(* IEC 61131-3 sources: weg-scada/M241_Bridge, 5 files *)

(* ---- POU_Diagnostics.st ---- *)
(*
  POU_Diagnostics - OPCIONAL

  Este programa es OPCIONAL. El M241 funciona como bridge transparente
  sin necesidad de programacion. Solo agregar este POU si se quiere
  monitorear el estado de comunicacion desde el PLC.

  Importar en Machine Expert: Project > Import > PLCOpen XML
  Asignar a MAST task si se usa.
*)

PROGRAM POU_Diagnostics
VAR
    (* Timers para detectar perdida de comunicacion *)
    tSSW1_Watchdog : TON;
    tSSW2_Watchdog : TON;

    (* Valores anteriores para detectar cambios *)
    wSSW1_PrevStatus : WORD := 16#FFFF;
    wSSW2_PrevStatus : WORD := 16#FFFF;

    (* Comunicacion OK flags *)
    bSSW1_Alive : BOOL;
    bSSW2_Alive : BOOL;

    (* Contadores de error *)
    udiSSW1_Errors : UDINT;
    udiSSW2_Errors : UDINT;

    (* LED output para diagnostico - usar salida digital del M241 *)
    bLED_AllOK     AT %QX0.0 : BOOL;  (* Q0 = Todos los esclavos OK *)
    bLED_SSW1_Fail AT %QX0.1 : BOOL;  (* Q1 = SSW1 sin comunicacion *)
    bLED_SSW2_Fail AT %QX0.2 : BOOL;  (* Q2 = SSW2 sin comunicacion *)
END_VAR

(* Detectar si SSW900 #1 esta respondiendo *)
(* Si el status word cambia, el esclavo esta vivo *)
IF GVL_SSW900.SSW1_StatusWord <> wSSW1_PrevStatus THEN
    wSSW1_PrevStatus := GVL_SSW900.SSW1_StatusWord;
    bSSW1_Alive := TRUE;
    tSSW1_Watchdog(IN := FALSE);  (* Reset timer *)
END_IF

tSSW1_Watchdog(IN := TRUE, PT := T#10S);
IF tSSW1_Watchdog.Q THEN
    bSSW1_Alive := FALSE;
    udiSSW1_Errors := udiSSW1_Errors + 1;
    tSSW1_Watchdog(IN := FALSE);
END_IF

(* Detectar si SSW900 #2 esta respondiendo *)
IF GVL_SSW900.SSW2_StatusWord <> wSSW2_PrevStatus THEN
    wSSW2_PrevStatus := GVL_SSW900.SSW2_StatusWord;
    bSSW2_Alive := TRUE;
    tSSW2_Watchdog(IN := FALSE);
END_IF

tSSW2_Watchdog(IN := TRUE, PT := T#10S);
IF tSSW2_Watchdog.Q THEN
    bSSW2_Alive := FALSE;
    udiSSW2_Errors := udiSSW2_Errors + 1;
    tSSW2_Watchdog(IN := FALSE);
END_IF

(* Actualizar variables globales *)
GVL_SSW900.SSW1_CommOK := bSSW1_Alive;
GVL_SSW900.SSW2_CommOK := bSSW2_Alive;
GVL_SSW900.SSW1_CommErrors := udiSSW1_Errors;
GVL_SSW900.SSW2_CommErrors := udiSSW2_Errors;

(* LEDs de diagnostico *)
bLED_AllOK := bSSW1_Alive AND bSSW2_Alive;
bLED_SSW1_Fail := NOT bSSW1_Alive;
bLED_SSW2_Fail := NOT bSSW2_Alive;

(* ---- WEG_Banner_Trending.st ---- *)
// ============================================================================
// WEG ALARM BANNER + TRENDING SUPPORT
// Single scrolling banner showing active faults from all 8 devices
// Trending buffer for WebVisu Trend element
// ============================================================================

// ============================================================================
// GVL: GVL_Banner (add to existing GVL_HMI or create separate)
// ============================================================================

{attribute 'qualified_only'}
VAR_GLOBAL

    // ---- Alarm Banner ----
    sBannerText         : STRING(255);      // Current text displayed in banner
    sBannerFull         : STRING(255);      // Full concatenated alarm string
    bBannerBlink        : BOOL;             // Blink flag for banner background
    iBannerColor        : INT;              // 0=No alarms(green), 1=Warning(yellow), 2=Fault(red)
    bHasFaults          : BOOL;             // At least one fault active

    // ---- Trending Data (WebVisu Trend uses these directly) ----
    // CFW900 Currents
    rTrend_CFW1_Current : REAL;
    rTrend_CFW2_Current : REAL;
    rTrend_CFW3_Current : REAL;
    rTrend_CFW4_Current : REAL;

    // CFW900 Frequencies
    rTrend_CFW1_Freq    : REAL;
    rTrend_CFW2_Freq    : REAL;
    rTrend_CFW3_Freq    : REAL;
    rTrend_CFW4_Freq    : REAL;

    // SSW900 Currents
    rTrend_SSW1_Current : REAL;
    rTrend_SSW2_Current : REAL;
    rTrend_SSW3_Current : REAL;
    rTrend_SSW4_Current : REAL;

END_VAR

// ============================================================================
// PROGRAM: PRG_AlarmBanner
// Builds a single scrolling text with all active faults
// Task: MAST
// ============================================================================

PROGRAM PRG_AlarmBanner
VAR
    i               : INT;
    sTemp           : STRING(255);
    iFaultCount     : INT;

    // Scroll control
    iScrollPos      : INT := 0;
    iScrollLen      : INT;
    tScrollTimer    : TON;
    tBlinkTimer     : TON;
    bBlinkState     : BOOL;

    // Rotation: cycle through faults one at a time
    iDisplayIndex   : INT := 0;         // Which fault to show (0..iFaultCount-1)
    tRotateTimer    : TON;
    aFaultMessages  : ARRAY[0..7] OF STRING(80);
    iFaultTotal     : INT;
END_VAR

// =========================================
// STEP 1: Collect all active faults
// =========================================
iFaultTotal := 0;

// Check CFW900 devices
FOR i := 1 TO 4 DO
    IF GVL_WEG.stCFW900[i].bFault THEN
        aFaultMessages[iFaultTotal] := CONCAT(
            CONCAT('CFW900#', INT_TO_STRING(i)),
            CONCAT(': ', FC_CFW900_FaultText(GVL_WEG.stCFW900[i].wFaultCode))
        );
        iFaultTotal := iFaultTotal + 1;

    ELSIF NOT GVL_WEG.stCFW900[i].bOnline AND GVL_WEG.stCFW900[i].uiCommErrCount > 5 THEN
        aFaultMessages[iFaultTotal] := CONCAT('CFW900#', CONCAT(INT_TO_STRING(i), ': COMM LOST'));
        iFaultTotal := iFaultTotal + 1;
    END_IF;
END_FOR;

// Check SSW900 devices
FOR i := 1 TO 4 DO
    IF GVL_WEG.stSSW900[i].bFault THEN
        aFaultMessages[iFaultTotal] := CONCAT(
            CONCAT('SSW900#', INT_TO_STRING(i)),
            CONCAT(': ', FC_SSW900_FaultText(GVL_WEG.stSSW900[i].wFaultCode))
        );
        iFaultTotal := iFaultTotal + 1;

    ELSIF NOT GVL_WEG.stSSW900[i].bOnline AND GVL_WEG.stSSW900[i].uiCommErrCount > 5 THEN
        aFaultMessages[iFaultTotal] := CONCAT('SSW900#', CONCAT(INT_TO_STRING(i), ': COMM LOST'));
        iFaultTotal := iFaultTotal + 1;
    END_IF;
END_FOR;

// =========================================
// STEP 2: Update banner state
// =========================================
GVL_Banner.bHasFaults := (iFaultTotal > 0);

IF iFaultTotal = 0 THEN
    // No faults - show OK message
    GVL_Banner.sBannerText := 'SYSTEM OK - All drives operating normally';
    GVL_Banner.iBannerColor := 0;       // Green
    GVL_Banner.bBannerBlink := FALSE;
    iDisplayIndex := 0;

ELSIF iFaultTotal = 1 THEN
    // Single fault - show it fixed (no rotation needed)
    GVL_Banner.sBannerText := CONCAT('!! ', CONCAT(aFaultMessages[0], ' !!'));
    GVL_Banner.iBannerColor := 2;       // Red
    GVL_Banner.bBannerBlink := TRUE;

ELSE
    // Multiple faults - rotate display every 3 seconds
    tRotateTimer(IN := TRUE, PT := T#3S);
    IF tRotateTimer.Q THEN
        tRotateTimer(IN := FALSE);
        iDisplayIndex := iDisplayIndex + 1;
        IF iDisplayIndex >= iFaultTotal THEN
            iDisplayIndex := 0;
        END_IF;
    END_IF;

    // Build display: "!! [2/3] CFW900#1: F002 Overcurrent !!"
    GVL_Banner.sBannerText := CONCAT(
        CONCAT('!! [', CONCAT(INT_TO_STRING(iDisplayIndex + 1), CONCAT('/', INT_TO_STRING(iFaultTotal)))),
        CONCAT('] ', CONCAT(aFaultMessages[iDisplayIndex], ' !!'))
    );
    GVL_Banner.iBannerColor := 2;       // Red
    GVL_Banner.bBannerBlink := TRUE;

END_IF;

// =========================================
// STEP 3: Blink control (500ms toggle)
// =========================================
tBlinkTimer(IN := NOT tBlinkTimer.Q, PT := T#500MS);
IF tBlinkTimer.Q THEN
    bBlinkState := NOT bBlinkState;
END_IF;

IF GVL_Banner.bBannerBlink THEN
    GVL_Banner.bBannerBlink := bBlinkState;    // Toggle for HMI animation
END_IF;

// ============================================================================
// PROGRAM: PRG_Trending
// Copies monitoring data to trending variables
// Task: MAST
// ============================================================================

PROGRAM PRG_Trending
VAR
END_VAR

// CFW900 Currents
GVL_Banner.rTrend_CFW1_Current := GVL_WEG.stCFW900[1].rOutputCurrent;
GVL_Banner.rTrend_CFW2_Current := GVL_WEG.stCFW900[2].rOutputCurrent;
GVL_Banner.rTrend_CFW3_Current := GVL_WEG.stCFW900[3].rOutputCurrent;
GVL_Banner.rTrend_CFW4_Current := GVL_WEG.stCFW900[4].rOutputCurrent;

// CFW900 Frequencies
GVL_Banner.rTrend_CFW1_Freq := GVL_WEG.stCFW900[1].rOutputFreq;
GVL_Banner.rTrend_CFW2_Freq := GVL_WEG.stCFW900[2].rOutputFreq;
GVL_Banner.rTrend_CFW3_Freq := GVL_WEG.stCFW900[3].rOutputFreq;
GVL_Banner.rTrend_CFW4_Freq := GVL_WEG.stCFW900[4].rOutputFreq;

// SSW900 Currents
GVL_Banner.rTrend_SSW1_Current := GVL_WEG.stSSW900[1].rMotorCurrent;
GVL_Banner.rTrend_SSW2_Current := GVL_WEG.stSSW900[2].rMotorCurrent;
GVL_Banner.rTrend_SSW3_Current := GVL_WEG.stSSW900[3].rMotorCurrent;
GVL_Banner.rTrend_SSW4_Current := GVL_WEG.stSSW900[4].rMotorCurrent;

(* ---- WEG_DataLog_Voltage.st ---- *)
// ============================================================================
// WEG DATA LOGGING (SD Card) + VOLTAGE EMPHASIS
// Exports CSV to M241 SD card + enhanced voltage monitoring
// Libraries required: FileIO, SysFile, SysTimeRtc, CAA File
// ============================================================================

// ============================================================================
// GVL: GVL_DataLog
// ============================================================================

{attribute 'qualified_only'}
VAR_GLOBAL

    // ---- Data Logging Control ----
    bLogEnabled         : BOOL := TRUE;     // Enable/disable logging from HMI
    bLogActive          : BOOL;             // Logging is running
    bLogError           : BOOL;             // File error occurred
    sLogStatus          : STRING(60);       // Status message for HMI
    iLogInterval        : INT := 5;         // Log interval in seconds (adjustable from HMI)
    ulRecordCount       : UDINT;            // Total records written

    // ---- File Management ----
    bNewFileDaily       : BOOL := TRUE;     // Create new file each day
    sCurrentFileName    : STRING(80);       // Current log file name
    bSDCardPresent      : BOOL;             // SD card detected
    ulFileSizeKB        : UDINT;            // Current file size

    // ---- Manual Export Trigger ----
    bExportSnapshot     : BOOL;             // Trigger single snapshot from HMI
    bExportDone         : BOOL;             // Snapshot saved confirmation

    // ---- Voltage Monitoring (Enhanced) ----
    // CFW900 Voltages
    stCFW_Voltage       : ARRAY[1..4] OF ST_VoltageMonitor;

    // SSW900 Voltages
    stSSW_Voltage       : ARRAY[1..4] OF ST_VoltageMonitor;

    // Voltage Alarms
    bVoltageAlarmActive : BOOL;             // Any voltage alarm
    iVoltageAlarmCount  : INT;

    // Voltage Thresholds (adjustable from HMI)
    rCFW_DCBus_High     : REAL := 750.0;    // DC Bus overvoltage threshold (V)
    rCFW_DCBus_Low      : REAL := 350.0;    // DC Bus undervoltage threshold (V)
    rSSW_Motor_High     : REAL := 480.0;    // Motor overvoltage threshold (V)
    rSSW_Motor_Low      : REAL := 400.0;    // Motor undervoltage threshold (V)
    rSSW_Imbalance_Max  : REAL := 5.0;      // Max voltage imbalance (%) between SSW units

    // Trending Voltage
    rTrend_CFW1_DCVoltage : REAL;
    rTrend_CFW2_DCVoltage : REAL;
    rTrend_CFW3_DCVoltage : REAL;
    rTrend_CFW4_DCVoltage : REAL;
    rTrend_SSW1_Voltage   : REAL;
    rTrend_SSW2_Voltage   : REAL;
    rTrend_SSW3_Voltage   : REAL;
    rTrend_SSW4_Voltage   : REAL;

END_VAR

// ============================================================================
// DUT: ST_VoltageMonitor
// ============================================================================

TYPE ST_VoltageMonitor :
STRUCT
    rVoltageNow     : REAL;         // Current voltage reading
    rVoltageMin     : REAL;         // Minimum since reset
    rVoltageMax     : REAL;         // Maximum since reset
    rVoltageAvg     : REAL;         // Running average

    // Alarms
    bOvervoltage    : BOOL;         // Above high threshold
    bUndervoltage   : BOOL;         // Below low threshold
    bAlarm          : BOOL;         // Any voltage alarm

    // Stats
    rDeviation      : REAL;         // Deviation from average (%)
    ulSampleCount   : UDINT;        // Samples for average calc
    rAccumulator    : LREAL;        // Sum for average (internal)
END_STRUCT
END_TYPE

// ============================================================================
// PROGRAM: PRG_VoltageMonitor
// Enhanced voltage tracking with min/max/avg and alarms
// Task: MAST
// ============================================================================

PROGRAM PRG_VoltageMonitor
VAR
    i               : INT;
    rAvgSSW         : REAL;         // Average voltage across all SSW units
    iOnlineSSW      : INT;
    bFirstScan      : BOOL := TRUE;
END_VAR

// =========================================
// Initialize min/max on first scan
// =========================================
IF bFirstScan THEN
    FOR i := 1 TO 4 DO
        GVL_DataLog.stCFW_Voltage[i].rVoltageMin := 9999.0;
        GVL_DataLog.stCFW_Voltage[i].rVoltageMax := 0.0;
        GVL_DataLog.stSSW_Voltage[i].rVoltageMin := 9999.0;
        GVL_DataLog.stSSW_Voltage[i].rVoltageMax := 0.0;
    END_FOR;
    bFirstScan := FALSE;
END_IF;

// =========================================
// CFW900: DC Bus Voltage monitoring
// =========================================
GVL_DataLog.iVoltageAlarmCount := 0;

FOR i := 1 TO 4 DO
    IF GVL_WEG.stCFW900[i].bOnline THEN

        GVL_DataLog.stCFW_Voltage[i].rVoltageNow := GVL_WEG.stCFW900[i].rDCBusVoltage;

        // Min / Max
        IF GVL_DataLog.stCFW_Voltage[i].rVoltageNow < GVL_DataLog.stCFW_Voltage[i].rVoltageMin THEN
            GVL_DataLog.stCFW_Voltage[i].rVoltageMin := GVL_DataLog.stCFW_Voltage[i].rVoltageNow;
        END_IF;
        IF GVL_DataLog.stCFW_Voltage[i].rVoltageNow > GVL_DataLog.stCFW_Voltage[i].rVoltageMax THEN
            GVL_DataLog.stCFW_Voltage[i].rVoltageMax := GVL_DataLog.stCFW_Voltage[i].rVoltageNow;
        END_IF;

        // Running average
        GVL_DataLog.stCFW_Voltage[i].ulSampleCount := GVL_DataLog.stCFW_Voltage[i].ulSampleCount + 1;
        GVL_DataLog.stCFW_Voltage[i].rAccumulator := GVL_DataLog.stCFW_Voltage[i].rAccumulator +
            REAL_TO_LREAL(GVL_DataLog.stCFW_Voltage[i].rVoltageNow);

        IF GVL_DataLog.stCFW_Voltage[i].ulSampleCount > 0 THEN
            GVL_DataLog.stCFW_Voltage[i].rVoltageAvg := LREAL_TO_REAL(
                GVL_DataLog.stCFW_Voltage[i].rAccumulator /
                UDINT_TO_LREAL(GVL_DataLog.stCFW_Voltage[i].ulSampleCount)
            );
        END_IF;

        // Overvoltage / Undervoltage alarms
        GVL_DataLog.stCFW_Voltage[i].bOvervoltage :=
            GVL_DataLog.stCFW_Voltage[i].rVoltageNow > GVL_DataLog.rCFW_DCBus_High;
        GVL_DataLog.stCFW_Voltage[i].bUndervoltage :=
            GVL_DataLog.stCFW_Voltage[i].rVoltageNow < GVL_DataLog.rCFW_DCBus_Low;
        GVL_DataLog.stCFW_Voltage[i].bAlarm :=
            GVL_DataLog.stCFW_Voltage[i].bOvervoltage OR GVL_DataLog.stCFW_Voltage[i].bUndervoltage;

        IF GVL_DataLog.stCFW_Voltage[i].bAlarm THEN
            GVL_DataLog.iVoltageAlarmCount := GVL_DataLog.iVoltageAlarmCount + 1;
        END_IF;

    END_IF;
END_FOR;

// =========================================
// SSW900: Motor Voltage monitoring
// =========================================
rAvgSSW := 0.0;
iOnlineSSW := 0;

FOR i := 1 TO 4 DO
    IF GVL_WEG.stSSW900[i].bOnline THEN

        GVL_DataLog.stSSW_Voltage[i].rVoltageNow := GVL_WEG.stSSW900[i].rMotorVoltage;

        // Min / Max
        IF GVL_DataLog.stSSW_Voltage[i].rVoltageNow < GVL_DataLog.stSSW_Voltage[i].rVoltageMin THEN
            GVL_DataLog.stSSW_Voltage[i].rVoltageMin := GVL_DataLog.stSSW_Voltage[i].rVoltageNow;
        END_IF;
        IF GVL_DataLog.stSSW_Voltage[i].rVoltageNow > GVL_DataLog.stSSW_Voltage[i].rVoltageMax THEN
            GVL_DataLog.stSSW_Voltage[i].rVoltageMax := GVL_DataLog.stSSW_Voltage[i].rVoltageNow;
        END_IF;

        // Running average
        GVL_DataLog.stSSW_Voltage[i].ulSampleCount := GVL_DataLog.stSSW_Voltage[i].ulSampleCount + 1;
        GVL_DataLog.stSSW_Voltage[i].rAccumulator := GVL_DataLog.stSSW_Voltage[i].rAccumulator +
            REAL_TO_LREAL(GVL_DataLog.stSSW_Voltage[i].rVoltageNow);

        IF GVL_DataLog.stSSW_Voltage[i].ulSampleCount > 0 THEN
            GVL_DataLog.stSSW_Voltage[i].rVoltageAvg := LREAL_TO_REAL(
                GVL_DataLog.stSSW_Voltage[i].rAccumulator /
                UDINT_TO_LREAL(GVL_DataLog.stSSW_Voltage[i].ulSampleCount)
            );
        END_IF;

        // Overvoltage / Undervoltage alarms
        GVL_DataLog.stSSW_Voltage[i].bOvervoltage :=
            GVL_DataLog.stSSW_Voltage[i].rVoltageNow > GVL_DataLog.rSSW_Motor_High;
        GVL_DataLog.stSSW_Voltage[i].bUndervoltage :=
            GVL_DataLog.stSSW_Voltage[i].rVoltageNow < GVL_DataLog.rSSW_Motor_Low;
        GVL_DataLog.stSSW_Voltage[i].bAlarm :=
            GVL_DataLog.stSSW_Voltage[i].bOvervoltage OR GVL_DataLog.stSSW_Voltage[i].bUndervoltage;

        IF GVL_DataLog.stSSW_Voltage[i].bAlarm THEN
            GVL_DataLog.iVoltageAlarmCount := GVL_DataLog.iVoltageAlarmCount + 1;
        END_IF;

        // Accumulate for imbalance calculation
        rAvgSSW := rAvgSSW + GVL_DataLog.stSSW_Voltage[i].rVoltageNow;
        iOnlineSSW := iOnlineSSW + 1;

    END_IF;
END_FOR;

// =========================================
// SSW900: Voltage imbalance detection
// =========================================
IF iOnlineSSW >= 2 THEN
    rAvgSSW := rAvgSSW / INT_TO_REAL(iOnlineSSW);

    FOR i := 1 TO 4 DO
        IF GVL_WEG.stSSW900[i].bOnline AND rAvgSSW > 0.0 THEN
            GVL_DataLog.stSSW_Voltage[i].rDeviation :=
                ABS(GVL_DataLog.stSSW_Voltage[i].rVoltageNow - rAvgSSW) / rAvgSSW * 100.0;

            // Flag if deviation exceeds threshold
            IF GVL_DataLog.stSSW_Voltage[i].rDeviation > GVL_DataLog.rSSW_Imbalance_Max THEN
                GVL_DataLog.stSSW_Voltage[i].bAlarm := TRUE;
                GVL_DataLog.iVoltageAlarmCount := GVL_DataLog.iVoltageAlarmCount + 1;
            END_IF;
        END_IF;
    END_FOR;
END_IF;

GVL_DataLog.bVoltageAlarmActive := (GVL_DataLog.iVoltageAlarmCount > 0);

// =========================================
// Update trending voltage variables
// =========================================
GVL_DataLog.rTrend_CFW1_DCVoltage := GVL_DataLog.stCFW_Voltage[1].rVoltageNow;
GVL_DataLog.rTrend_CFW2_DCVoltage := GVL_DataLog.stCFW_Voltage[2].rVoltageNow;
GVL_DataLog.rTrend_CFW3_DCVoltage := GVL_DataLog.stCFW_Voltage[3].rVoltageNow;
GVL_DataLog.rTrend_CFW4_DCVoltage := GVL_DataLog.stCFW_Voltage[4].rVoltageNow;
GVL_DataLog.rTrend_SSW1_Voltage   := GVL_DataLog.stSSW_Voltage[1].rVoltageNow;
GVL_DataLog.rTrend_SSW2_Voltage   := GVL_DataLog.stSSW_Voltage[2].rVoltageNow;
GVL_DataLog.rTrend_SSW3_Voltage   := GVL_DataLog.stSSW_Voltage[3].rVoltageNow;
GVL_DataLog.rTrend_SSW4_Voltage   := GVL_DataLog.stSSW_Voltage[4].rVoltageNow;

// ============================================================================
// PROGRAM: PRG_DataLogger
// Writes CSV records to M241 SD card
// Task: MAST
// Libraries: CAA File (SysFile), SysTimeRtc
// ============================================================================

PROGRAM PRG_DataLogger
VAR
    // State machine
    iStep           : INT := 0;

    // Timer for log interval
    tLogInterval    : TON;
    tLogPT          : TIME;

    // File handling
    hFile           : CAA.FILE.FILE_HANDLE := CAA.FILE.INVALID_HANDLE;
    fbFileOpen      : CAA.FILE.Open;
    fbFileWrite     : CAA.FILE.Write;
    fbFileClose     : CAA.FILE.Close;

    // Date/Time
    dtCurrent       : DT;
    stTime          : TIMESTRUCT;
    sDate           : STRING(12);
    sTime           : STRING(10);
    sFileName       : STRING(80);

    // CSV building
    sCSVHeader      : STRING(255);
    sCSVLine        : STRING(255);
    sCSVLine2       : STRING(255);      // Continuation (long line)
    sTemp           : STRING(20);

    // State tracking
    iLastDay        : INT := -1;
    bHeaderWritten  : BOOL;
    bWriteError     : BOOL;
    i               : INT;
END_VAR

// =========================================
// Build log interval from HMI setting
// =========================================
tLogPT := INT_TO_TIME(GVL_DataLog.iLogInterval * 1000);

CASE iStep OF

    0: // ---- CHECK IF LOGGING ENABLED ----
        IF NOT GVL_DataLog.bLogEnabled THEN
            GVL_DataLog.bLogActive := FALSE;
            GVL_DataLog.sLogStatus := 'Logging disabled';
            RETURN;
        END_IF;

        GVL_DataLog.bLogActive := TRUE;
        iStep := 5;

    5: // ---- GET CURRENT DATE/TIME ----
        dtCurrent := GET_DATETIME();
        stTime := DT_TO_TIMESTRUCT(dtCurrent);

        // Build date string YYYY-MM-DD
        sDate := CONCAT(
            CONCAT(INT_TO_STRING(stTime.wYear), '-'),
            CONCAT(FC_PadZero(stTime.wMonth), CONCAT('-', FC_PadZero(stTime.wDay)))
        );

        // Build time string HH:MM:SS
        sTime := CONCAT(
            CONCAT(FC_PadZero(stTime.wHour), ':'),
            CONCAT(FC_PadZero(stTime.wMinute), CONCAT(':', FC_PadZero(stTime.wSecond)))
        );

        // Build filename: /sd0/WEG_LOG_2026-03-30.csv
        sFileName := CONCAT('/sd0/WEG_LOG_', CONCAT(sDate, '.csv'));
        GVL_DataLog.sCurrentFileName := sFileName;

        // Check if new day = new file
        IF INT_TO_INT(stTime.wDay) <> iLastDay THEN
            iLastDay := INT_TO_INT(stTime.wDay);
            bHeaderWritten := FALSE;
        END_IF;

        iStep := 10;

    10: // ---- WAIT FOR LOG INTERVAL ----
        tLogInterval(IN := TRUE, PT := tLogPT);

        // Also check for manual snapshot trigger
        IF tLogInterval.Q OR GVL_DataLog.bExportSnapshot THEN
            tLogInterval(IN := FALSE);
            GVL_DataLog.bExportSnapshot := FALSE;
            iStep := 20;
        END_IF;

    20: // ---- OPEN FILE (APPEND MODE) ----
        fbFileOpen(
            sFileName   := sFileName,
            eFileMode   := CAA.FILE.MODE.MRDWR,    // Read/Write (append)
            xExclusive  := FALSE
        );

        IF fbFileOpen.xDone THEN
            hFile := fbFileOpen.hFile;
            GVL_DataLog.bLogError := FALSE;

            IF NOT bHeaderWritten THEN
                iStep := 25;    // Write header first
            ELSE
                iStep := 30;    // Skip to data
            END_IF;

        ELSIF fbFileOpen.xError THEN
            // File might not exist, try create
            GVL_DataLog.bLogError := TRUE;
            GVL_DataLog.sLogStatus := 'SD Card error - check card';
            iStep := 10;
        END_IF;

    25: // ---- WRITE CSV HEADER ----
        sCSVHeader := 'DateTime,';
        sCSVHeader := CONCAT(sCSVHeader, 'CFW1_A,CFW1_Hz,CFW1_VDC,CFW1_Torq,CFW1_RPM,CFW1_Sts,');
        sCSVHeader := CONCAT(sCSVHeader, 'CFW2_A,CFW2_Hz,CFW2_VDC,CFW2_Torq,CFW2_RPM,CFW2_Sts,');
        sCSVHeader := CONCAT(sCSVHeader, 'CFW3_A,CFW3_Hz,CFW3_VDC,CFW3_Torq,CFW3_RPM,CFW3_Sts,');

        fbFileWrite(
            hFile   := hFile,
            pBuffer := ADR(sCSVHeader),
            szSize  := INT_TO_UDINT(LEN(sCSVHeader))
        );

        // Second part of header (line too long for single STRING)
        sCSVLine := 'CFW4_A,CFW4_Hz,CFW4_VDC,CFW4_Torq,CFW4_RPM,CFW4_Sts,';
        sCSVLine := CONCAT(sCSVLine, 'SSW1_A,SSW1_V,SSW1_kW,SSW1_Sts,');
        sCSVLine := CONCAT(sCSVLine, 'SSW2_A,SSW2_V,SSW2_kW,SSW2_Sts,');
        sCSVLine := CONCAT(sCSVLine, 'SSW3_A,SSW3_V,SSW3_kW,SSW3_Sts,');
        sCSVLine := CONCAT(sCSVLine, 'SSW4_A,SSW4_V,SSW4_kW,SSW4_Sts$N');

        fbFileWrite(
            hFile   := hFile,
            pBuffer := ADR(sCSVLine),
            szSize  := INT_TO_UDINT(LEN(sCSVLine))
        );

        bHeaderWritten := TRUE;
        iStep := 30;

    30: // ---- BUILD CSV DATA LINE ----
        // DateTime + CFW900 #1-#2
        sCSVLine := CONCAT(sDate, CONCAT(' ', CONCAT(sTime, ',')));

        FOR i := 1 TO 2 DO
            sCSVLine := CONCAT(sCSVLine,
                CONCAT(REAL_TO_STRING(GVL_WEG.stCFW900[i].rOutputCurrent), CONCAT(',',
                CONCAT(REAL_TO_STRING(GVL_WEG.stCFW900[i].rOutputFreq), CONCAT(',',
                CONCAT(REAL_TO_STRING(GVL_WEG.stCFW900[i].rDCBusVoltage), CONCAT(',',
                CONCAT(REAL_TO_STRING(GVL_WEG.stCFW900[i].rMotorTorque), CONCAT(',',
                CONCAT(REAL_TO_STRING(GVL_WEG.stCFW900[i].rSpeedRPM), CONCAT(',',
                CONCAT(WORD_TO_STRING(GVL_WEG.stCFW900[i].wStatusWord), ',')
                ))))))))))
            );
        END_FOR;

        // CFW900 #3-#4
        sCSVLine2 := '';
        FOR i := 3 TO 4 DO
            sCSVLine2 := CONCAT(sCSVLine2,
                CONCAT(REAL_TO_STRING(GVL_WEG.stCFW900[i].rOutputCurrent), CONCAT(',',
                CONCAT(REAL_TO_STRING(GVL_WEG.stCFW900[i].rOutputFreq), CONCAT(',',
                CONCAT(REAL_TO_STRING(GVL_WEG.stCFW900[i].rDCBusVoltage), CONCAT(',',
                CONCAT(REAL_TO_STRING(GVL_WEG.stCFW900[i].rMotorTorque), CONCAT(',',
                CONCAT(REAL_TO_STRING(GVL_WEG.stCFW900[i].rSpeedRPM), CONCAT(',',
                CONCAT(WORD_TO_STRING(GVL_WEG.stCFW900[i].wStatusWord), ',')
                ))))))))))
            );
        END_FOR;

        // SSW900 #1-#4
        FOR i := 1 TO 4 DO
            sCSVLine2 := CONCAT(sCSVLine2,
                CONCAT(REAL_TO_STRING(GVL_WEG.stSSW900[i].rMotorCurrent), CONCAT(',',
                CONCAT(REAL_TO_STRING(GVL_WEG.stSSW900[i].rMotorVoltage), CONCAT(',',
                CONCAT(REAL_TO_STRING(GVL_WEG.stSSW900[i].rMotorPower), CONCAT(',',
                CONCAT(WORD_TO_STRING(GVL_WEG.stSSW900[i].wStatusWord), ',')
                ))))))
            );
        END_FOR;
        sCSVLine2 := CONCAT(sCSVLine2, '$N');   // Newline

        iStep := 40;

    40: // ---- WRITE DATA TO FILE ----
        fbFileWrite(
            hFile   := hFile,
            pBuffer := ADR(sCSVLine),
            szSize  := INT_TO_UDINT(LEN(sCSVLine))
        );
        fbFileWrite(
            hFile   := hFile,
            pBuffer := ADR(sCSVLine2),
            szSize  := INT_TO_UDINT(LEN(sCSVLine2))
        );

        GVL_DataLog.ulRecordCount := GVL_DataLog.ulRecordCount + 1;
        GVL_DataLog.bExportDone := TRUE;
        GVL_DataLog.sLogStatus := CONCAT('Logging OK - Records: ', UDINT_TO_STRING(GVL_DataLog.ulRecordCount));

        iStep := 50;

    50: // ---- CLOSE FILE ----
        fbFileClose(hFile := hFile);

        IF fbFileClose.xDone THEN
            hFile := CAA.FILE.INVALID_HANDLE;
            iStep := 10;   // Back to wait
        END_IF;

END_CASE;

// ============================================================================
// FUNCTION: FC_PadZero
// Pads single digit to 2 chars: 5 -> '05'
// ============================================================================

FUNCTION FC_PadZero : STRING(3)
VAR_INPUT
    wValue : WORD;
END_VAR

IF wValue < 10 THEN
    FC_PadZero := CONCAT('0', WORD_TO_STRING(wValue));
ELSE
    FC_PadZero := WORD_TO_STRING(wValue);
END_IF;

// ============================================================================
// FUNCTION: FC_ResetVoltageStats
// Call from HMI button to reset min/max/avg
// ============================================================================

FUNCTION FC_ResetVoltageStats : BOOL
VAR
    i : INT;
END_VAR

FOR i := 1 TO 4 DO
    GVL_DataLog.stCFW_Voltage[i].rVoltageMin := 9999.0;
    GVL_DataLog.stCFW_Voltage[i].rVoltageMax := 0.0;
    GVL_DataLog.stCFW_Voltage[i].rVoltageAvg := 0.0;
    GVL_DataLog.stCFW_Voltage[i].rAccumulator := 0.0;
    GVL_DataLog.stCFW_Voltage[i].ulSampleCount := 0;

    GVL_DataLog.stSSW_Voltage[i].rVoltageMin := 9999.0;
    GVL_DataLog.stSSW_Voltage[i].rVoltageMax := 0.0;
    GVL_DataLog.stSSW_Voltage[i].rVoltageAvg := 0.0;
    GVL_DataLog.stSSW_Voltage[i].rAccumulator := 0.0;
    GVL_DataLog.stSSW_Voltage[i].ulSampleCount := 0;
END_FOR;

FC_ResetVoltageStats := TRUE;

(* ---- WEG_HMI_Support.st ---- *)
// ============================================================================
// WEG HMI SUPPORT CODE - WebVisu (Machine Expert)
// Variables and logic to support the HMI visualization screens
// ============================================================================

// ============================================================================
// GVL: GVL_HMI
// Variables used by WebVisu screens
// ============================================================================

{attribute 'qualified_only'}
VAR_GLOBAL

    // ---- Navigation ----
    iActivePage         : INT := 0;         // 0=Overview, 1=CFW Detail, 2=SSW Detail
    iSelectedCFW        : INT := 1;         // Selected CFW900 (1..4) for detail view
    iSelectedSSW        : INT := 1;         // Selected SSW900 (1..4) for detail view

    // ---- Overview: CFW900 summary bars (scaled 0-100%) ----
    arCFW_CurrentPct    : ARRAY[1..4] OF REAL;  // Current as % of nominal
    arCFW_FreqPct       : ARRAY[1..4] OF REAL;  // Frequency as % of nominal
    arCFW_StatusColor   : ARRAY[1..4] OF INT;   // 0=Off, 1=Ready, 2=Running, 3=Fault

    // ---- Overview: SSW900 summary bars ----
    arSSW_CurrentPct    : ARRAY[1..4] OF REAL;
    arSSW_StatusColor   : ARRAY[1..4] OF INT;   // 0=Off, 1=Ready, 2=Running/Bypass, 3=Starting, 4=Fault

    // ---- Detail: CFW900 selected device ----
    stCFW_Detail        : ST_CFW900_HMI_Detail;

    // ---- Detail: SSW900 selected device ----
    stSSW_Detail        : ST_SSW900_HMI_Detail;

    // ---- Alarms ----
    bAlarmActive        : BOOL;             // Any alarm active
    iAlarmCount         : INT;              // Number of active alarms
    asAlarmText         : ARRAY[1..8] OF STRING(80);  // Alarm texts for each device

    // ---- CFW900 Nominal Values (adjust to your motors) ----
    rCFW_NominalCurrent : REAL := 25.0;     // Nominal current (A) - ADJUST
    rCFW_NominalFreq    : REAL := 60.0;     // Nominal frequency (Hz) - ADJUST

    // ---- SSW900 Nominal Values ----
    rSSW_NominalCurrent : REAL := 50.0;     // Nominal current (A) - ADJUST

END_VAR

// ============================================================================
// DUT: ST_CFW900_HMI_Detail
// ============================================================================

TYPE ST_CFW900_HMI_Detail :
STRUCT
    sDeviceName     : STRING(30);
    rSpeedRPM       : REAL;
    rCurrent        : REAL;
    rFrequency      : REAL;
    rDCBusVoltage   : REAL;
    rTorque         : REAL;
    sFaultText      : STRING(40);
    sStatusText     : STRING(20);
    iStatusColor    : INT;          // For color animation
    bOnline         : BOOL;
    uiCommErrors    : UINT;

    // Bar graph values (0-100%)
    rCurrentBar     : REAL;
    rFreqBar        : REAL;
    rTorqueBar      : REAL;
    rVoltageBar     : REAL;
END_STRUCT
END_TYPE

// ============================================================================
// DUT: ST_SSW900_HMI_Detail
// ============================================================================

TYPE ST_SSW900_HMI_Detail :
STRUCT
    sDeviceName     : STRING(30);
    rCurrent        : REAL;
    rVoltage        : REAL;
    rPower          : REAL;
    sFaultText      : STRING(40);
    sStatusText     : STRING(20);
    iStatusColor    : INT;
    bOnline         : BOOL;
    uiCommErrors    : UINT;

    // Bar graph values (0-100%)
    rCurrentBar     : REAL;
    rVoltageBar     : REAL;
    rPowerBar       : REAL;
END_STRUCT
END_TYPE

// ============================================================================
// PROGRAM: PRG_HMI_Update
// Updates all HMI variables from raw Modbus data
// Task: MAST
// ============================================================================

PROGRAM PRG_HMI_Update
VAR
    i : INT;
END_VAR

// =========================================
// OVERVIEW: Update CFW900 bars and colors
// =========================================
FOR i := 1 TO 4 DO

    // Current as percentage of nominal
    IF GVL_HMI.rCFW_NominalCurrent > 0.0 THEN
        GVL_HMI.arCFW_CurrentPct[i] := (GVL_WEG.stCFW900[i].rOutputCurrent / GVL_HMI.rCFW_NominalCurrent) * 100.0;
    END_IF;

    // Frequency as percentage of nominal
    IF GVL_HMI.rCFW_NominalFreq > 0.0 THEN
        GVL_HMI.arCFW_FreqPct[i] := (GVL_WEG.stCFW900[i].rOutputFreq / GVL_HMI.rCFW_NominalFreq) * 100.0;
    END_IF;

    // Status color: 0=Gray(Off), 1=Green(Ready), 2=Blue(Running), 3=Red(Fault)
    IF GVL_WEG.stCFW900[i].bFault THEN
        GVL_HMI.arCFW_StatusColor[i] := 3;
    ELSIF GVL_WEG.stCFW900[i].bRunning THEN
        GVL_HMI.arCFW_StatusColor[i] := 2;
    ELSIF GVL_WEG.stCFW900[i].bReady THEN
        GVL_HMI.arCFW_StatusColor[i] := 1;
    ELSE
        GVL_HMI.arCFW_StatusColor[i] := 0;
    END_IF;

END_FOR;

// =========================================
// OVERVIEW: Update SSW900 bars and colors
// =========================================
FOR i := 1 TO 4 DO

    IF GVL_HMI.rSSW_NominalCurrent > 0.0 THEN
        GVL_HMI.arSSW_CurrentPct[i] := (GVL_WEG.stSSW900[i].rMotorCurrent / GVL_HMI.rSSW_NominalCurrent) * 100.0;
    END_IF;

    // 0=Gray, 1=Green(Ready), 2=Blue(Running), 3=Yellow(Starting), 4=Red(Fault)
    IF GVL_WEG.stSSW900[i].bFault THEN
        GVL_HMI.arSSW_StatusColor[i] := 4;
    ELSIF GVL_WEG.stSSW900[i].bRunning THEN
        GVL_HMI.arSSW_StatusColor[i] := 2;
    ELSIF GVL_WEG.stSSW900[i].bStarting THEN
        GVL_HMI.arSSW_StatusColor[i] := 3;
    ELSIF GVL_WEG.stSSW900[i].bReady THEN
        GVL_HMI.arSSW_StatusColor[i] := 1;
    ELSE
        GVL_HMI.arSSW_StatusColor[i] := 0;
    END_IF;

END_FOR;

// =========================================
// DETAIL: Update CFW900 detail view
// =========================================
IF GVL_HMI.iSelectedCFW >= 1 AND GVL_HMI.iSelectedCFW <= 4 THEN

    i := GVL_HMI.iSelectedCFW;

    GVL_HMI.stCFW_Detail.sDeviceName   := CONCAT('CFW900 #', INT_TO_STRING(i));
    GVL_HMI.stCFW_Detail.rSpeedRPM     := GVL_WEG.stCFW900[i].rSpeedRPM;
    GVL_HMI.stCFW_Detail.rCurrent      := GVL_WEG.stCFW900[i].rOutputCurrent;
    GVL_HMI.stCFW_Detail.rFrequency    := GVL_WEG.stCFW900[i].rOutputFreq;
    GVL_HMI.stCFW_Detail.rDCBusVoltage := GVL_WEG.stCFW900[i].rDCBusVoltage;
    GVL_HMI.stCFW_Detail.rTorque       := GVL_WEG.stCFW900[i].rMotorTorque;
    GVL_HMI.stCFW_Detail.bOnline       := GVL_WEG.stCFW900[i].bOnline;
    GVL_HMI.stCFW_Detail.uiCommErrors  := GVL_WEG.stCFW900[i].uiCommErrCount;
    GVL_HMI.stCFW_Detail.iStatusColor  := GVL_HMI.arCFW_StatusColor[i];

    // Bar graphs (capped at 120%)
    GVL_HMI.stCFW_Detail.rCurrentBar  := LIMIT(0.0, GVL_HMI.arCFW_CurrentPct[i], 120.0);
    GVL_HMI.stCFW_Detail.rFreqBar     := LIMIT(0.0, GVL_HMI.arCFW_FreqPct[i], 120.0);
    GVL_HMI.stCFW_Detail.rTorqueBar   := LIMIT(0.0, GVL_WEG.stCFW900[i].rMotorTorque, 120.0);
    GVL_HMI.stCFW_Detail.rVoltageBar  := LIMIT(0.0, GVL_WEG.stCFW900[i].rDCBusVoltage / 7.0, 120.0);

    // Status text
    IF GVL_WEG.stCFW900[i].bFault THEN
        GVL_HMI.stCFW_Detail.sStatusText := 'FAULT';
    ELSIF GVL_WEG.stCFW900[i].bRunning THEN
        GVL_HMI.stCFW_Detail.sStatusText := 'RUNNING';
    ELSIF GVL_WEG.stCFW900[i].bReady THEN
        GVL_HMI.stCFW_Detail.sStatusText := 'READY';
    ELSE
        GVL_HMI.stCFW_Detail.sStatusText := 'OFF';
    END_IF;

    // Fault text
    GVL_HMI.stCFW_Detail.sFaultText := FC_CFW900_FaultText(GVL_WEG.stCFW900[i].wFaultCode);

END_IF;

// =========================================
// DETAIL: Update SSW900 detail view
// =========================================
IF GVL_HMI.iSelectedSSW >= 1 AND GVL_HMI.iSelectedSSW <= 4 THEN

    i := GVL_HMI.iSelectedSSW;

    GVL_HMI.stSSW_Detail.sDeviceName   := CONCAT('SSW900 #', INT_TO_STRING(i));
    GVL_HMI.stSSW_Detail.rCurrent      := GVL_WEG.stSSW900[i].rMotorCurrent;
    GVL_HMI.stSSW_Detail.rVoltage      := GVL_WEG.stSSW900[i].rMotorVoltage;
    GVL_HMI.stSSW_Detail.rPower        := GVL_WEG.stSSW900[i].rMotorPower;
    GVL_HMI.stSSW_Detail.bOnline       := GVL_WEG.stSSW900[i].bOnline;
    GVL_HMI.stSSW_Detail.uiCommErrors  := GVL_WEG.stSSW900[i].uiCommErrCount;
    GVL_HMI.stSSW_Detail.iStatusColor  := GVL_HMI.arSSW_StatusColor[i];

    // Bar graphs
    GVL_HMI.stSSW_Detail.rCurrentBar := LIMIT(0.0, GVL_HMI.arSSW_CurrentPct[i], 120.0);
    GVL_HMI.stSSW_Detail.rVoltageBar := LIMIT(0.0, GVL_WEG.stSSW900[i].rMotorVoltage / 5.0, 120.0);
    GVL_HMI.stSSW_Detail.rPowerBar   := LIMIT(0.0, GVL_WEG.stSSW900[i].rMotorPower / 1.0, 120.0);

    // Status text
    IF GVL_WEG.stSSW900[i].bFault THEN
        GVL_HMI.stSSW_Detail.sStatusText := 'FAULT';
    ELSIF GVL_WEG.stSSW900[i].bRunning THEN
        GVL_HMI.stSSW_Detail.sStatusText := 'RUNNING';
    ELSIF GVL_WEG.stSSW900[i].bStarting THEN
        GVL_HMI.stSSW_Detail.sStatusText := 'STARTING';
    ELSIF GVL_WEG.stSSW900[i].bReady THEN
        GVL_HMI.stSSW_Detail.sStatusText := 'READY';
    ELSE
        GVL_HMI.stSSW_Detail.sStatusText := 'OFF';
    END_IF;

    GVL_HMI.stSSW_Detail.sFaultText := FC_SSW900_FaultText(GVL_WEG.stSSW900[i].wFaultCode);

END_IF;

// =========================================
// ALARMS: Update alarm summary
// =========================================
GVL_HMI.iAlarmCount := 0;
GVL_HMI.bAlarmActive := FALSE;

FOR i := 1 TO 4 DO
    IF GVL_WEG.stCFW900[i].bFault THEN
        GVL_HMI.iAlarmCount := GVL_HMI.iAlarmCount + 1;
        GVL_HMI.bAlarmActive := TRUE;
        GVL_HMI.asAlarmText[i] := CONCAT(CONCAT('CFW900 #', INT_TO_STRING(i)),
            CONCAT(' - FAULT: ', FC_CFW900_FaultText(GVL_WEG.stCFW900[i].wFaultCode)));
    ELSIF NOT GVL_WEG.stCFW900[i].bOnline THEN
        GVL_HMI.iAlarmCount := GVL_HMI.iAlarmCount + 1;
        GVL_HMI.bAlarmActive := TRUE;
        GVL_HMI.asAlarmText[i] := CONCAT('CFW900 #', CONCAT(INT_TO_STRING(i), ' - COMM LOST'));
    ELSE
        GVL_HMI.asAlarmText[i] := '';
    END_IF;
END_FOR;

FOR i := 1 TO 4 DO
    IF GVL_WEG.stSSW900[i].bFault THEN
        GVL_HMI.iAlarmCount := GVL_HMI.iAlarmCount + 1;
        GVL_HMI.bAlarmActive := TRUE;
        GVL_HMI.asAlarmText[i + 4] := CONCAT(CONCAT('SSW900 #', INT_TO_STRING(i)),
            CONCAT(' - FAULT: ', FC_SSW900_FaultText(GVL_WEG.stSSW900[i].wFaultCode)));
    ELSIF NOT GVL_WEG.stSSW900[i].bOnline THEN
        GVL_HMI.iAlarmCount := GVL_HMI.iAlarmCount + 1;
        GVL_HMI.bAlarmActive := TRUE;
        GVL_HMI.asAlarmText[i + 4] := CONCAT('SSW900 #', CONCAT(INT_TO_STRING(i), ' - COMM LOST'));
    ELSE
        GVL_HMI.asAlarmText[i + 4] := '';
    END_IF;
END_FOR;

// ============================================================================
// FUNCTION: FC_CFW900_FaultText
// Returns fault description from CFW900 fault code
// ============================================================================

FUNCTION FC_CFW900_FaultText : STRING(40)
VAR_INPUT
    wFaultCode : WORD;
END_VAR

CASE WORD_TO_INT(wFaultCode) OF
    0:  FC_CFW900_FaultText := 'No Fault';
    2:  FC_CFW900_FaultText := 'F002: Overcurrent';
    3:  FC_CFW900_FaultText := 'F003: DC Link Overvoltage';
    4:  FC_CFW900_FaultText := 'F004: IGBT Overtemp';
    5:  FC_CFW900_FaultText := 'F005: Motor Overload';
    6:  FC_CFW900_FaultText := 'F006: Drive Overtemp';
    7:  FC_CFW900_FaultText := 'F007: Overcurrent Phase U';
    8:  FC_CFW900_FaultText := 'F008: Overcurrent Phase V';
    9:  FC_CFW900_FaultText := 'F009: Overcurrent Phase W';
    12: FC_CFW900_FaultText := 'F012: Phase Loss Input';
    21: FC_CFW900_FaultText := 'F021: Earth Fault';
    22: FC_CFW900_FaultText := 'F022: Motor Overtemp PTC';
    33: FC_CFW900_FaultText := 'F033: Undervoltage';
    49: FC_CFW900_FaultText := 'F049: Motor Stalled';
    70: FC_CFW900_FaultText := 'F070: Communication Error';
    72: FC_CFW900_FaultText := 'F072: Fieldbus Timeout';
    74: FC_CFW900_FaultText := 'F074: Serial Comm Error';
ELSE
    FC_CFW900_FaultText := CONCAT('Fault Code: ', WORD_TO_STRING(wFaultCode));
END_CASE;

// ============================================================================
// FUNCTION: FC_SSW900_FaultText
// Returns fault description from SSW900 fault code
// ============================================================================

FUNCTION FC_SSW900_FaultText : STRING(40)
VAR_INPUT
    wFaultCode : WORD;
END_VAR

CASE WORD_TO_INT(wFaultCode) OF
    0:  FC_SSW900_FaultText := 'No Fault';
    1:  FC_SSW900_FaultText := 'F01: Motor Overcurrent';
    2:  FC_SSW900_FaultText := 'F02: Phase Sequence';
    3:  FC_SSW900_FaultText := 'F03: Phase Loss Input';
    4:  FC_SSW900_FaultText := 'F04: Phase Loss Output';
    5:  FC_SSW900_FaultText := 'F05: Thyristor Short';
    6:  FC_SSW900_FaultText := 'F06: Heatsink Overtemp';
    7:  FC_SSW900_FaultText := 'F07: Motor Overload';
    8:  FC_SSW900_FaultText := 'F08: Undervoltage';
    9:  FC_SSW900_FaultText := 'F09: Overvoltage';
    10: FC_SSW900_FaultText := 'F10: Phase Imbalance';
    11: FC_SSW900_FaultText := 'F11: Motor PTC Overtemp';
    20: FC_SSW900_FaultText := 'F20: Bypass Contactor';
    30: FC_SSW900_FaultText := 'F30: Communication Error';
    51: FC_SSW900_FaultText := 'F51: Locked Rotor';
    73: FC_SSW900_FaultText := 'F73: Serial Timeout';
ELSE
    FC_SSW900_FaultText := CONCAT('Fault Code: ', WORD_TO_STRING(wFaultCode));
END_CASE;

(* ---- WEG_ModbusTCP_Map.st ---- *)
// ============================================================================
// PRG_ModbusTCP_Map
// Maps GVL_WEG variables to %MW registers for Node-RED access
// Add to MAST task AFTER PRG_WEG_Modbus_SL1 and PRG_WEG_Modbus_SL2
// ============================================================================

PROGRAM PRG_ModbusTCP_Map
VAR
    i       : INT;
    iBase   : INT;
END_VAR

// =========================================
// CFW900 -> %MW0 to %MW39 (4 devices x 10 registers)
// =========================================
FOR i := 1 TO 4 DO
    iBase := (i - 1) * 10;

    %MW[iBase + 0]  := WORD_TO_INT(GVL_WEG.stCFW900[i].wStatusWord);
    %MW[iBase + 1]  := REAL_TO_INT(GVL_WEG.stCFW900[i].rSpeedRPM);
    %MW[iBase + 2]  := REAL_TO_INT(GVL_WEG.stCFW900[i].rOutputCurrent * 10.0);
    %MW[iBase + 3]  := REAL_TO_INT(GVL_WEG.stCFW900[i].rOutputFreq * 10.0);
    %MW[iBase + 4]  := REAL_TO_INT(GVL_WEG.stCFW900[i].rDCBusVoltage * 10.0);
    %MW[iBase + 5]  := REAL_TO_INT(GVL_WEG.stCFW900[i].rMotorTorque * 10.0);
    %MW[iBase + 6]  := WORD_TO_INT(GVL_WEG.stCFW900[i].wFaultCode);
    %MW[iBase + 7]  := BOOL_TO_INT(GVL_WEG.stCFW900[i].bOnline);
    %MW[iBase + 8]  := UINT_TO_INT(GVL_WEG.stCFW900[i].uiCommErrCount);
    %MW[iBase + 9]  := 0;  // Reserved
END_FOR;

// =========================================
// SSW900 -> %MW40 to %MW79 (4 devices x 10 registers)
// =========================================
FOR i := 1 TO 4 DO
    iBase := 40 + (i - 1) * 10;

    %MW[iBase + 0]  := WORD_TO_INT(GVL_WEG.stSSW900[i].wStatusWord);
    %MW[iBase + 1]  := REAL_TO_INT(GVL_WEG.stSSW900[i].rMotorCurrent * 10.0);
    %MW[iBase + 2]  := REAL_TO_INT(GVL_WEG.stSSW900[i].rMotorVoltage * 10.0);
    %MW[iBase + 3]  := REAL_TO_INT(GVL_WEG.stSSW900[i].rMotorPower * 10.0);
    %MW[iBase + 4]  := WORD_TO_INT(GVL_WEG.stSSW900[i].wFaultCode);
    %MW[iBase + 5]  := BOOL_TO_INT(GVL_WEG.stSSW900[i].bOnline);
    %MW[iBase + 6]  := UINT_TO_INT(GVL_WEG.stSSW900[i].uiCommErrCount);
    %MW[iBase + 7]  := 0;
    %MW[iBase + 8]  := 0;
    %MW[iBase + 9]  := 0;
END_FOR;
